FUNCTION_BLOCK PAEActFlap2 EXTENDS PAEActuator2way
VAR_INPUT
END_VAR
VAR_OUTPUT
END_VAR
VAR
END_VAR

METHOD PUBLIC PAEActFlap2
VAR_INPUT
END_VAR
END_METHOD

END_FUNCTION_BLOCK

(* stored: Version 1.1.0.1, ProductVersion 3.1.4020.12
   POU PAEActFlap2: Id {d3d11179-ed49-4ee7-8d42-35700e302c65}, SpecialFunc None
   Method PAEActFlap2: Id {98e3c9a7-959f-4900-81ef-4b9281b6958a} *)
